// Mitsubishi GX Works2 project: PLC_7_27.11_watch   PLC: FX3G

// global labels: Global1
VAR_GLOBAL CONSTANT
  Const_flickers : REAL := 5;
END_VAR
VAR_GLOBAL
  SW_start_day AT X010 : BOOL;
  LI_active_day AT Y010 : BOOL;
  RE_init_org AT D1100 : REAL;
  RE_init_pml AT D1105 : REAL;
  RE_init_clm AT D1110 : REAL;
  RE_wash_org AT D1130 : REAL;
  RE_wash_pml AT D1135 : REAL;
  RE_wash_clm AT D1140 : REAL;
  RE_squeeze AT D1145 : REAL;
  RE_juice AT D1150 : REAL;
  RE_storage AT D1155 : REAL;
  SW_emeragnce AT X007 : BOOL;
  SW_start_wash AT X002 : BOOL;
  LI_active_wash AT Y005 : BOOL;
  SW_col_fruits AT X001 : BOOL;
  LI_active_col AT Y001 : BOOL;
  SW_start_squeeze AT X011 : BOOL;
  LI_flicker_1 AT Y002 : BOOL;
  LI_flicker_2 AT Y003 : BOOL;
  SW_qa AT X003 : BOOL;
END_VAR
VAR_GLOBAL CONSTANT
  Const_min_Range : INT := 1;
  Const_max_Range : INT := 5;
END_VAR
VAR_GLOBAL
  LI_qa AT Y004 : BOOL;
  Analog_output AT D8282 : REAL;
END_VAR
VAR_GLOBAL CONSTANT
  Const_ratio_2 : REAL := 2;
END_VAR
VAR_GLOBAL
  HL_3_sec_stop AT M0 : BOOL;
  HL_blink1 AT M1 : BOOL;
  HL_first_init AT M2 : BOOL;
END_VAR
VAR_GLOBAL CONSTANT
  Const_min_fruit : REAL := 1;
END_VAR
VAR_GLOBAL
  HL_min_fruit AT M3 : BOOL;
  HL_first_check AT M4 : BOOL;
END_VAR
VAR_GLOBAL CONSTANT
  Const_timer_3 : INT := 30;
END_VAR
VAR_GLOBAL
  TC_timer_3 AT TC3 : BOOL;
  TS_timer_3 AT TS3 : BOOL;
  HL_blink2 AT M5 : BOOL;
  HL_blink3 AT M6 : BOOL;
  TC_blink1 AT TC1 : BOOL;
  TS_blink1 AT TS1 : BOOL;
  TC_blink2 AT TC2 : BOOL;
  TS_blink2 AT TS2 : BOOL;
  TN_timer_3 AT TN3 : INT;
  TN_blink1 AT TN1 : INT;
  HL_stop_day AT M7 : BOOL;
  HL_start_wash AT M8 : BOOL;
  HL_active_day AT M9 : BOOL;
  RE_buffer AT D1170 : REAL;
END_VAR
VAR_GLOBAL CONSTANT
  Const_max_org : REAL := 50;
END_VAR
VAR_GLOBAL
  RE_half_amount AT D1175 : REAL;
  HL_end_station_1 AT M11 : BOOL;
  HL_reset_day AT M12 : BOOL;
  HL_start_squeeze AT M13 : BOOL;
  HL_blink_end AT M14 : BOOL;
  HL_end_station_3 AT M15 : BOOL;
  HL_end_station_2 AT M16 : BOOL;
  HL_end_station_4 AT M17 : BOOL;
  RE_analog_input AT D8201 : INT;
  HL_min_range AT M18 : BOOL;
  HL_max_range AT M19 : BOOL;
  HL_start_station_4 AT M20 : BOOL;
  RE_timer_generic AT D1185 : INT;
END_VAR
VAR_GLOBAL CONSTANT
  Const_timer_5 : INT := 50;
END_VAR
VAR_GLOBAL
  HL_help_check AT M21 : BOOL;
  HL_bad_test AT M22 : BOOL;
  CC_counter AT CC0 : BOOL;
END_VAR
VAR_GLOBAL CONSTANT
  Const_counter : INT := 2;
END_VAR
VAR_GLOBAL
  CS_counter AT CS0 : BOOL;
  HL_garbge AT M23 : BOOL;
  Analog_Input AT D8281 : INT;
  RE_div_to_normal AT D1190 : REAL;
END_VAR
VAR_GLOBAL CONSTANT
  Const_200 : INT := 200;
  Const_400 : INT := 400;
END_VAR
VAR_GLOBAL
  HL_check_wash1 AT M24 : BOOL;
  HL_check_wash2 AT M25 : BOOL;
  SW_start_donation AT X005 : BOOL;
  LI_donation1 AT Y006 : BOOL;
  RE_donation AT D1200 : REAL;
  RE_donation_org AT D1205 : INT;
  RE_donation_clm AT D1210 : INT;
  RE_donation_pml AT D1215 : INT;
  RE_donation_org_real AT D1220 : REAL;
  RE_donation_clm_real AT D1225 : REAL;
  RE_donation_pml_real AT D1230 : REAL;
END_VAR
VAR_GLOBAL CONSTANT
  Const_0 : REAL;
END_VAR
VAR_GLOBAL
  HL_donation_remain AT M26 : BOOL;
  LI_donation2 AT Y007 : BOOL;
END_VAR
VAR_GLOBAL CONSTANT
  Const_min_storage : INT := 150;
  Const_max_storage : INT := 300;
END_VAR
VAR_GLOBAL
  HL_end_station_0 AT M27 : BOOL;
END_VAR
VAR_GLOBAL CONSTANT
  Const_range_0 : REAL := 9472;
  Const_range_1 : REAL := 9475;
  Const_range_2 : REAL := 9476;
END_VAR
VAR_GLOBAL
  RE_range : ARRAY [0..2] OF BOOL;
  HL_storage_range0 AT M100 : BOOL;
  HL_storage_range1 AT M101 : BOOL;
  HL_storage_range2 AT M102 : BOOL;
  RE_storage_int AT D1232 : INT;
  HL_end_indicator_station_0 AT M103 : BOOL;
  CN_counter AT CN0 : INT;
END_VAR
VAR_GLOBAL CONSTANT
  Const_timer_03 : INT := 3;
  Const_ratio_2_modulo : INT := 2;
END_VAR

// task Task_01 (event TRUE, interval 0, priority 31): POU_01

PROGRAM POU_01
(* structured ladder/FBD written out as ST: instructions are called as NAME(EN, inputs, outputs); _pN, _eN, _tN stand for wires *)
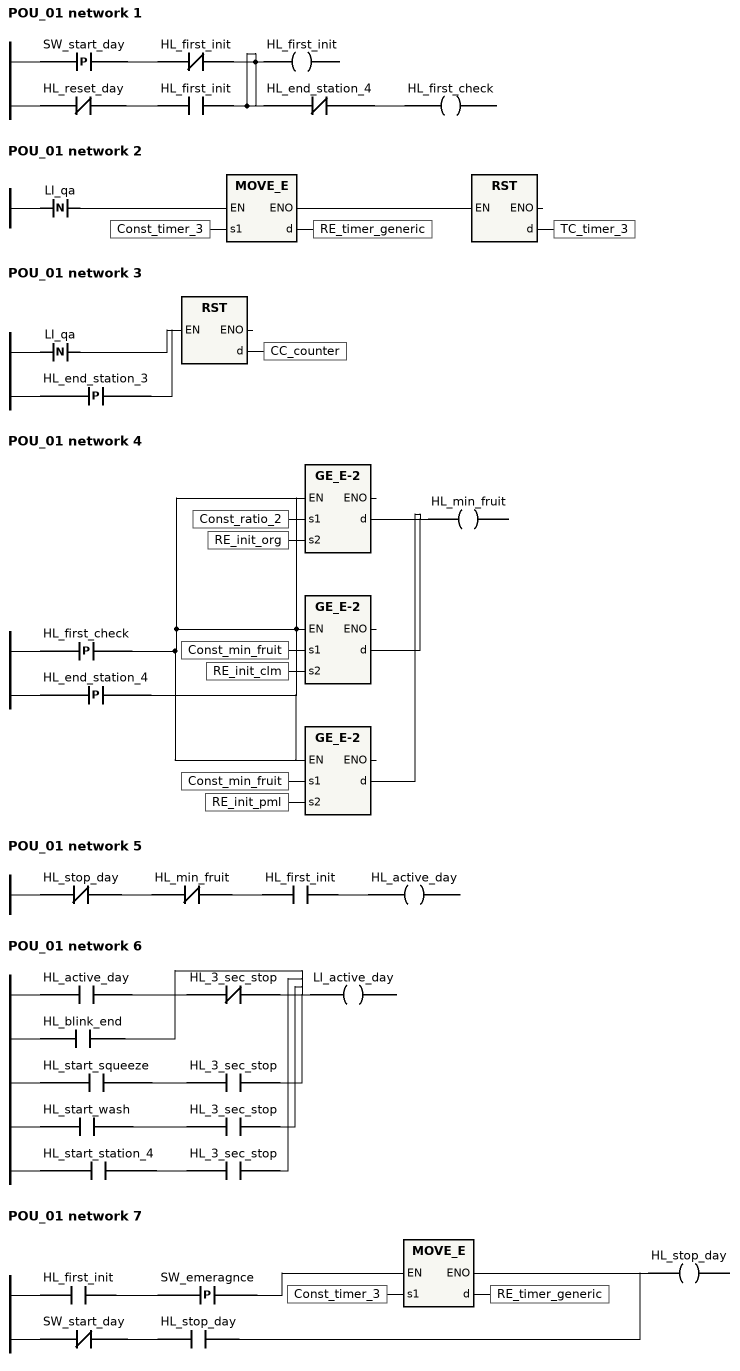
(* network 1 *)
_p1 := (LDP(TRUE, SW_start_day) AND NOT HL_first_init) OR (NOT HL_reset_day AND HL_first_init);
HL_first_init := _p1;
HL_first_check := _p1 AND NOT HL_end_station_4;
(* network 2 *)
_e1 := MOVE_E(LDF(TRUE, LI_qa), Const_timer_3, RE_timer_generic);
RST(_e1, TC_timer_3);
(* network 3 *)
RST(LDF(TRUE, LI_qa) OR LDP(TRUE, HL_end_station_3), CC_counter);
(* network 4 *)
_p1 := LDP(TRUE, HL_first_check) OR LDP(TRUE, HL_end_station_4);
GE_E(_p1, Const_ratio_2, RE_init_org, _t2);
GE_E(_p1, Const_min_fruit, RE_init_clm, _t3);
GE_E(_p1, Const_min_fruit, RE_init_pml, _t4);
HL_min_fruit := _t2 OR _t3 OR _t4;
(* network 5 *)
HL_active_day := NOT HL_stop_day AND NOT HL_min_fruit AND HL_first_init;
(* network 6 *)
LI_active_day := (HL_active_day AND NOT HL_3_sec_stop) OR HL_blink_end OR (HL_start_squeeze AND HL_3_sec_stop) OR (HL_start_wash AND HL_3_sec_stop) OR (HL_start_station_4 AND HL_3_sec_stop);
(* network 7 *)
_e1 := MOVE_E(HL_first_init AND LDP(TRUE, SW_emeragnce), Const_timer_3, RE_timer_generic);
HL_stop_day := _e1 OR (NOT SW_start_day AND HL_stop_day);
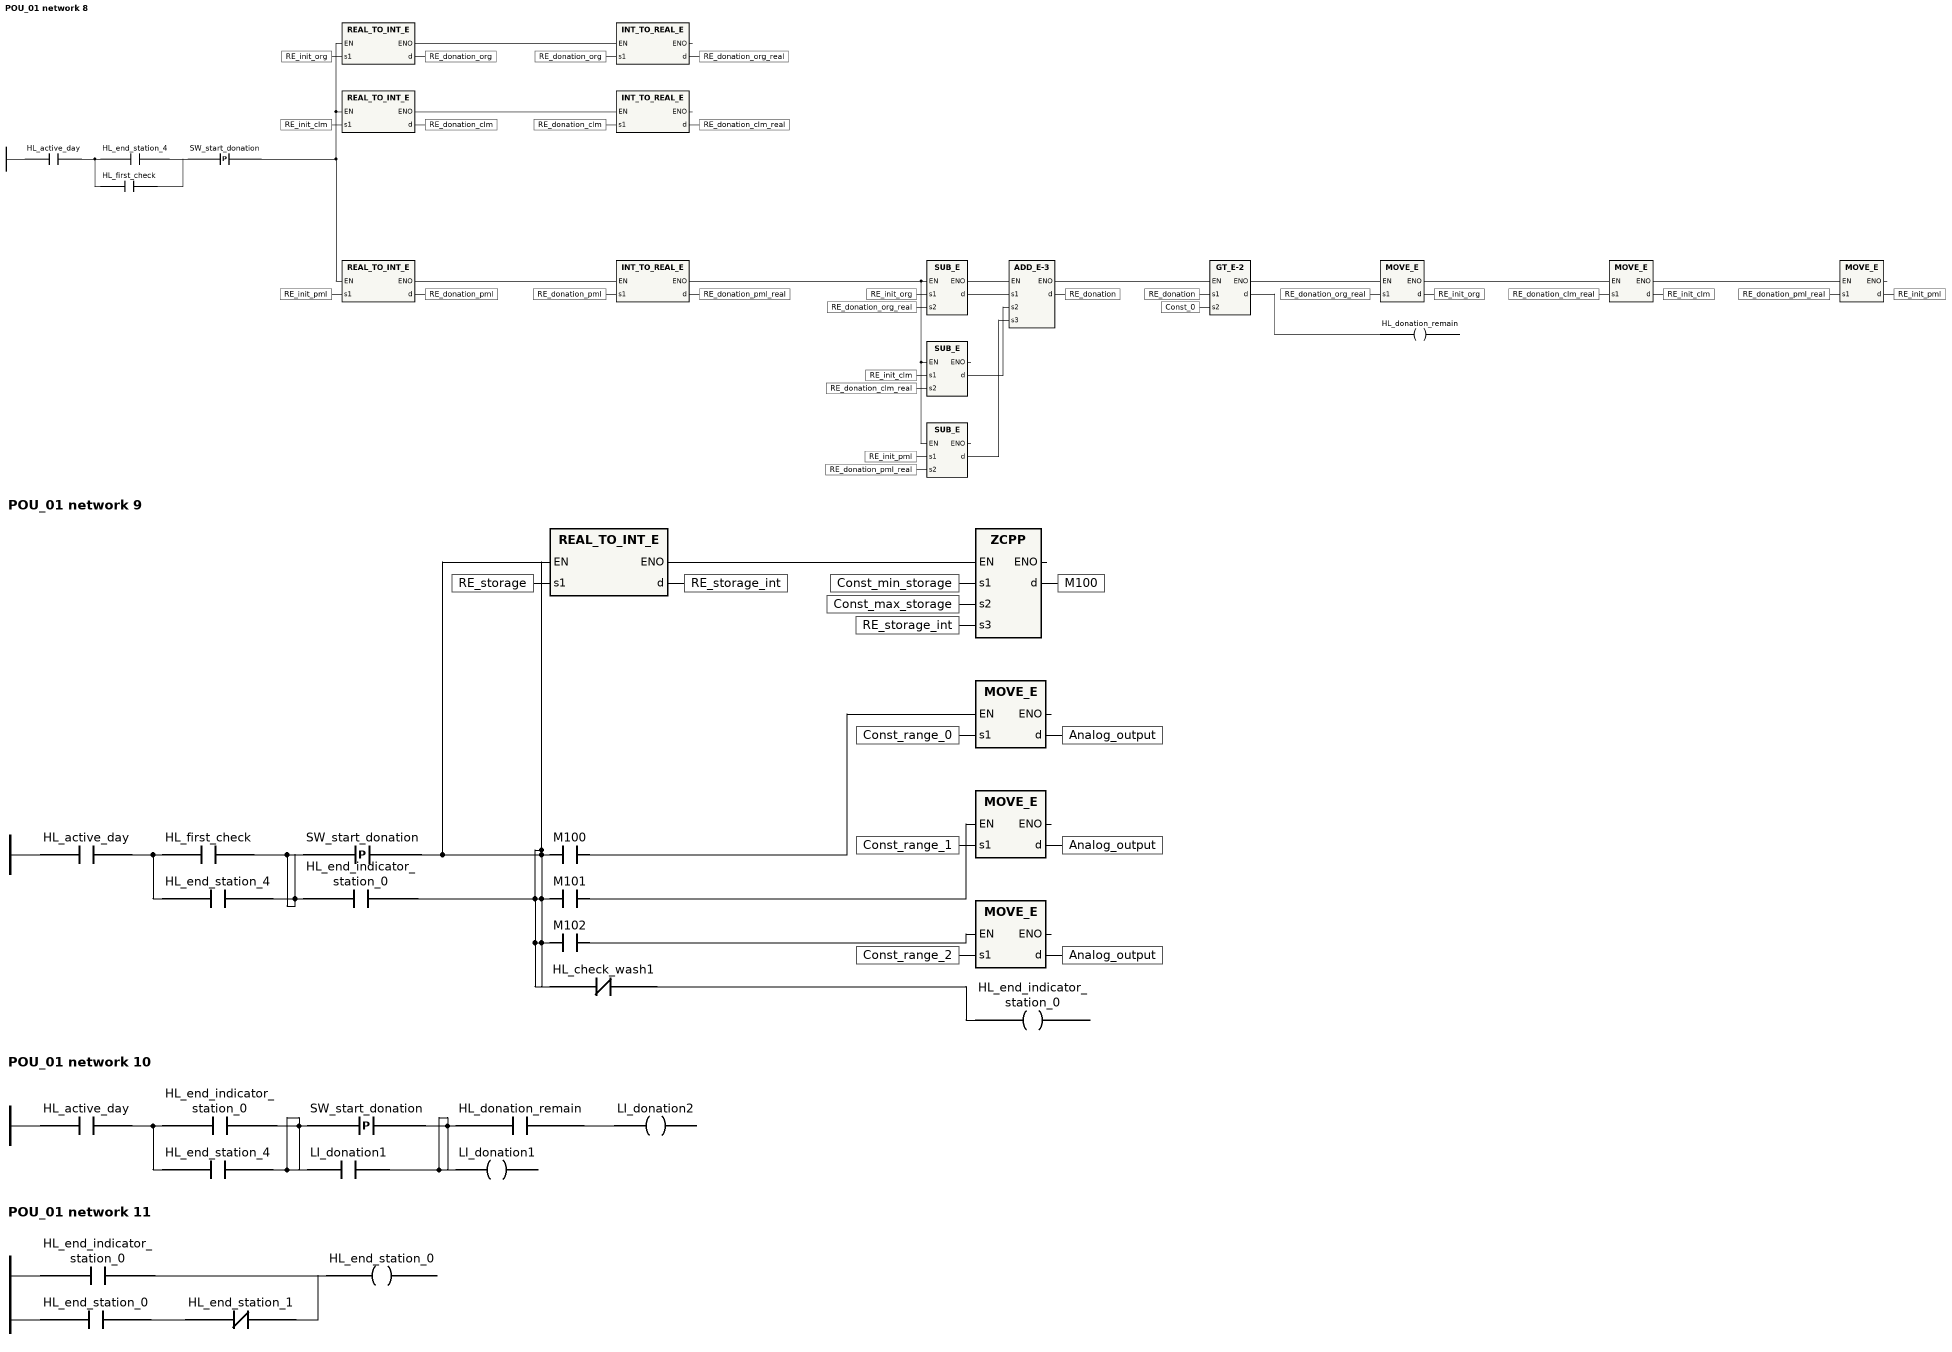
(* network 8 *)
_p1 := ((HL_active_day AND HL_end_station_4) OR (HL_active_day AND HL_first_check)) AND LDP(TRUE, SW_start_donation);
_e2 := REAL_TO_INT_E(_p1, RE_init_org, RE_donation_org);
INT_TO_REAL_E(_e2, RE_donation_org, RE_donation_org_real);
_e3 := REAL_TO_INT_E(_p1, RE_init_clm, RE_donation_clm);
INT_TO_REAL_E(_e3, RE_donation_clm, RE_donation_clm_real);
_e4 := REAL_TO_INT_E(_p1, RE_init_pml, RE_donation_pml);
_e5 := INT_TO_REAL_E(_e4, RE_donation_pml, RE_donation_pml_real);
_e7 := SUB_E(_e5, RE_init_org, RE_donation_org_real, _t6);
SUB_E(_e5, RE_init_clm, RE_donation_clm_real, _t8);
SUB_E(_e5, RE_init_pml, RE_donation_pml_real, _t9);
_e10 := ADD_E(_e7, _t6, _t8, _t9, RE_donation);
_e12 := GT_E(_e10, RE_donation, Const_0, _t11);
HL_donation_remain := _t11;
_e13 := MOVE_E(_e12, RE_donation_org_real, RE_init_org);
_e14 := MOVE_E(_e13, RE_donation_clm_real, RE_init_clm);
MOVE_E(_e14, RE_donation_pml_real, RE_init_pml);
(* network 9 *)
_p1 := (HL_active_day AND HL_first_check) OR (HL_active_day AND HL_end_station_4);
_p2 := (_p1 AND LDP(TRUE, SW_start_donation)) OR (_p1 AND HL_end_indicator_station_0);
_e3 := REAL_TO_INT_E(_p2, RE_storage, RE_storage_int);
ZCPP(_e3, Const_min_storage, Const_max_storage, RE_storage_int, M100);
MOVE_E(_p2 AND M100, Const_range_0, Analog_output);
MOVE_E(_p2 AND M101, Const_range_1, Analog_output);
MOVE_E(_p2 AND M102, Const_range_2, Analog_output);
HL_end_indicator_station_0 := _p2 AND NOT HL_check_wash1;
(* network 10 *)
_p1 := (HL_active_day AND HL_end_indicator_station_0) OR (HL_active_day AND HL_end_station_4);
_p2 := (_p1 AND LDP(TRUE, SW_start_donation)) OR (_p1 AND LI_donation1);
LI_donation2 := _p2 AND HL_donation_remain;
LI_donation1 := _p2;
(* network 11 *)
HL_end_station_0 := HL_end_indicator_station_0 OR (HL_end_station_0 AND NOT HL_end_station_1);
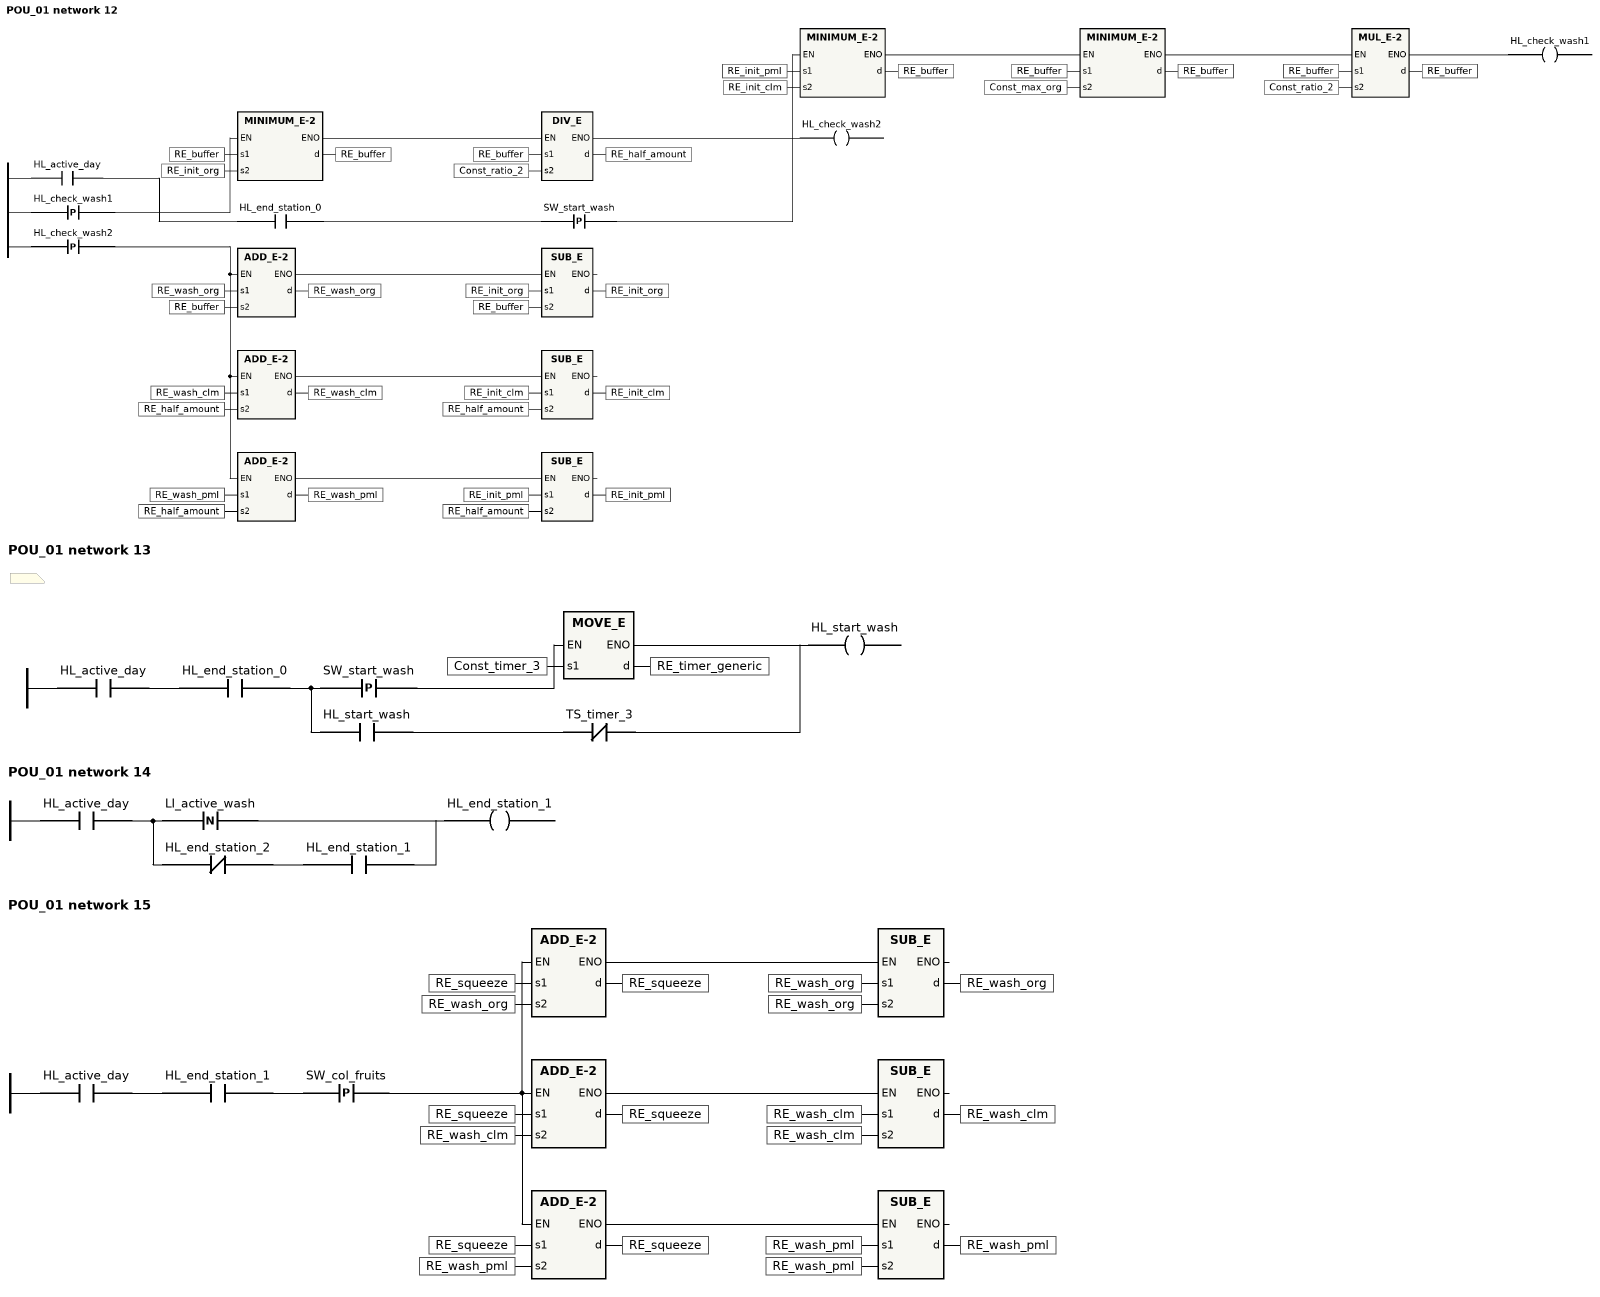
(* network 12 *)
_e1 := MINIMUM_E(HL_active_day AND HL_end_station_0 AND LDP(TRUE, SW_start_wash), RE_init_pml, RE_init_clm, RE_buffer);
_e2 := MINIMUM_E(_e1, RE_buffer, Const_max_org, RE_buffer);
_e3 := MUL_E(_e2, RE_buffer, Const_ratio_2, RE_buffer);
HL_check_wash1 := _e3;
_e4 := MINIMUM_E(LDP(TRUE, HL_check_wash1), RE_buffer, RE_init_org, RE_buffer);
_e5 := DIV_E(_e4, RE_buffer, Const_ratio_2, RE_half_amount);
HL_check_wash2 := _e5;
_p6 := LDP(TRUE, HL_check_wash2);
_e7 := ADD_E(_p6, RE_wash_org, RE_buffer, RE_wash_org);
SUB_E(_e7, RE_init_org, RE_buffer, RE_init_org);
_e8 := ADD_E(_p6, RE_wash_clm, RE_half_amount, RE_wash_clm);
SUB_E(_e8, RE_init_clm, RE_half_amount, RE_init_clm);
_e9 := ADD_E(_p6, RE_wash_pml, RE_half_amount, RE_wash_pml);
SUB_E(_e9, RE_init_pml, RE_half_amount, RE_init_pml);
(* network 13 *)
(*  *)
_p1 := HL_active_day AND HL_end_station_0;
_e2 := MOVE_E(_p1 AND LDP(TRUE, SW_start_wash), Const_timer_3, RE_timer_generic);
HL_start_wash := _e2 OR (_p1 AND HL_start_wash AND NOT TS_timer_3);
(* network 14 *)
HL_end_station_1 := (HL_active_day AND LDF(TRUE, LI_active_wash)) OR (HL_active_day AND NOT HL_end_station_2 AND HL_end_station_1);
(* network 15 *)
_p1 := HL_active_day AND HL_end_station_1 AND LDP(TRUE, SW_col_fruits);
_e2 := ADD_E(_p1, RE_squeeze, RE_wash_org, RE_squeeze);
SUB_E(_e2, RE_wash_org, RE_wash_org, RE_wash_org);
_e3 := ADD_E(_p1, RE_squeeze, RE_wash_clm, RE_squeeze);
SUB_E(_e3, RE_wash_clm, RE_wash_clm, RE_wash_clm);
_e4 := ADD_E(_p1, RE_squeeze, RE_wash_pml, RE_squeeze);
SUB_E(_e4, RE_wash_pml, RE_wash_pml, RE_wash_pml);
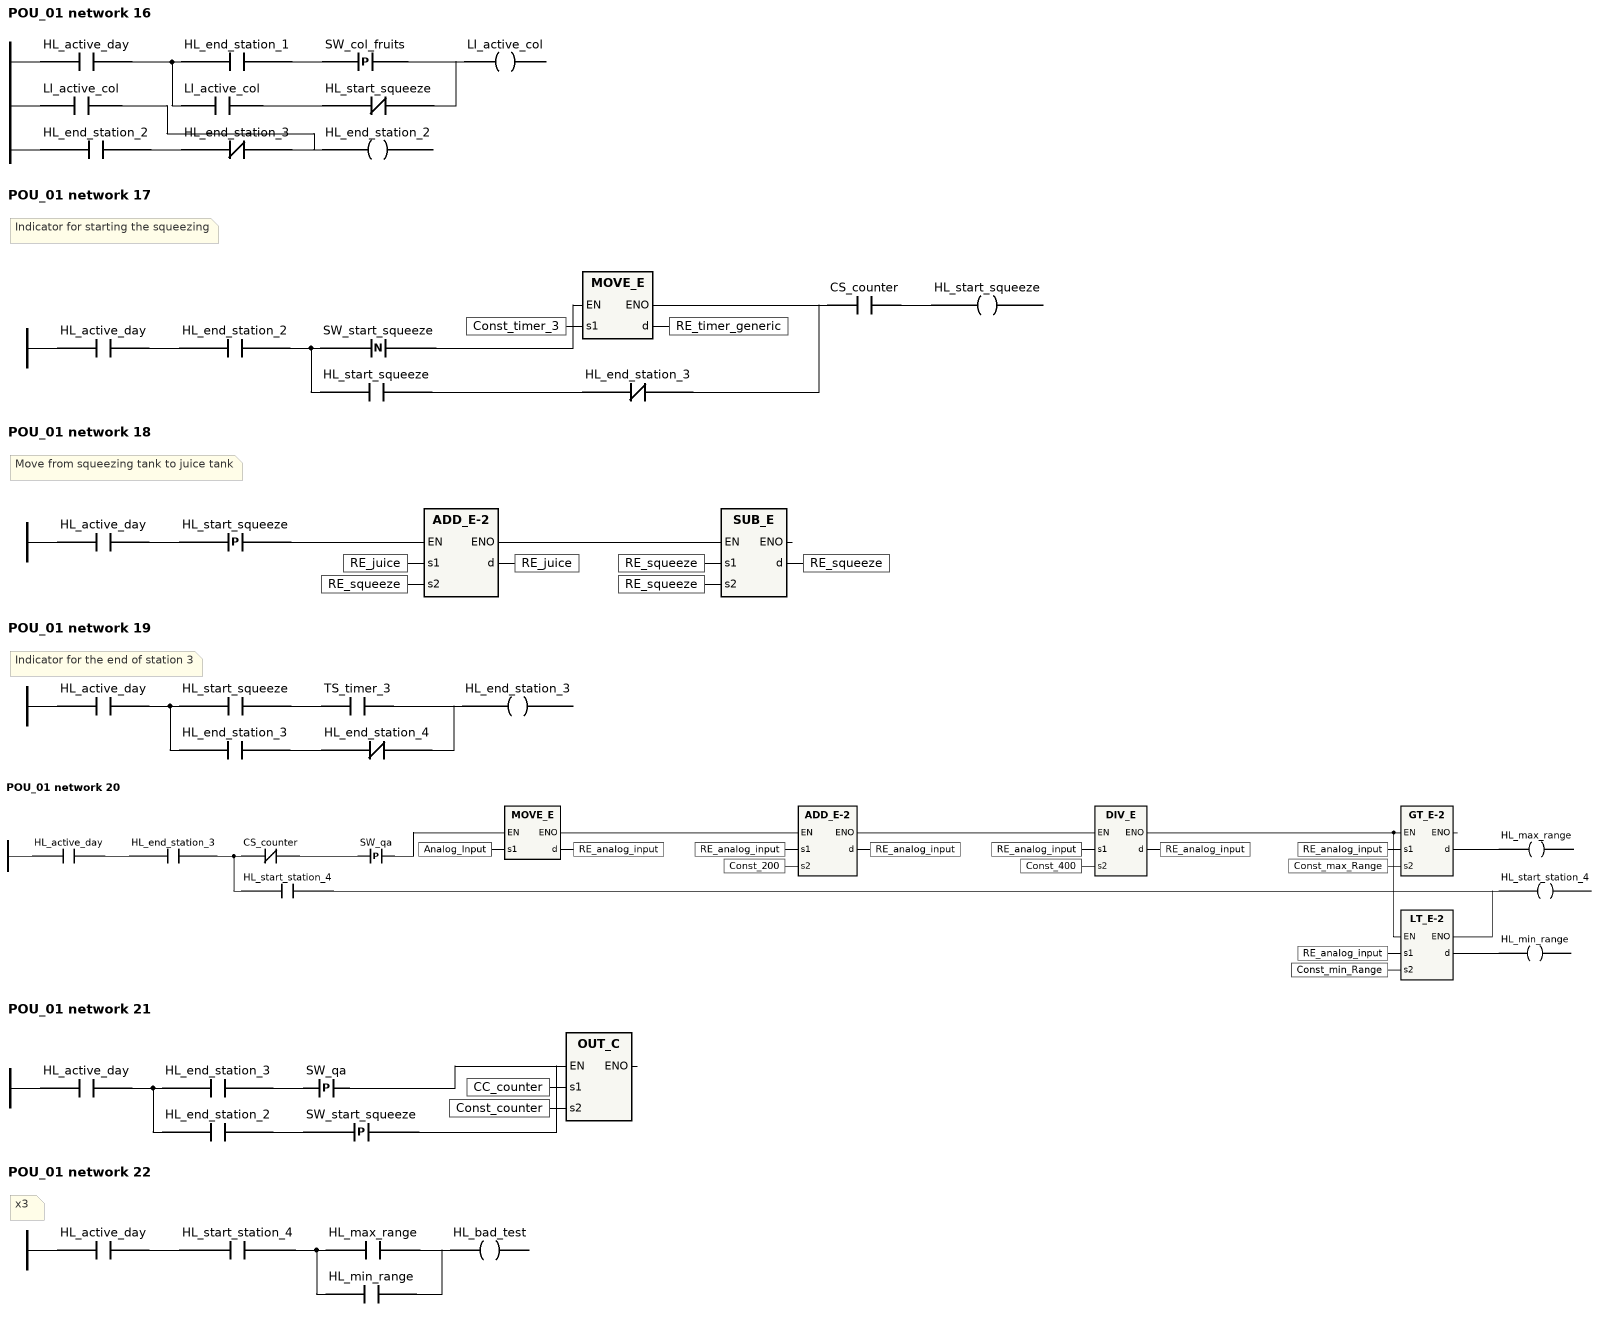
(* network 16 *)
LI_active_col := (HL_active_day AND HL_end_station_1 AND LDP(TRUE, SW_col_fruits)) OR (HL_active_day AND LI_active_col AND NOT HL_start_squeeze);
HL_end_station_2 := LI_active_col OR (HL_end_station_2 AND NOT HL_end_station_3);
(* network 17 *)
(* Indicator for starting the squeezing *)
_p1 := HL_active_day AND HL_end_station_2;
_e2 := MOVE_E(_p1 AND LDF(TRUE, SW_start_squeeze), Const_timer_3, RE_timer_generic);
HL_start_squeeze := (_e2 OR (_p1 AND HL_start_squeeze AND NOT HL_end_station_3)) AND CS_counter;
(* network 18 *)
(* Move from squeezing tank to juice tank *)
_e1 := ADD_E(HL_active_day AND LDP(TRUE, HL_start_squeeze), RE_juice, RE_squeeze, RE_juice);
SUB_E(_e1, RE_squeeze, RE_squeeze, RE_squeeze);
(* network 19 *)
(* Indicator for the end of station 3 *)
HL_end_station_3 := (HL_active_day AND HL_start_squeeze AND TS_timer_3) OR (HL_active_day AND HL_end_station_3 AND NOT HL_end_station_4);
(* network 20 *)
_p1 := HL_active_day AND HL_end_station_3;
_e2 := MOVE_E(_p1 AND NOT CS_counter AND LDP(TRUE, SW_qa), Analog_Input, RE_analog_input);
_e3 := ADD_E(_e2, RE_analog_input, Const_200, RE_analog_input);
_e4 := DIV_E(_e3, RE_analog_input, Const_400, RE_analog_input);
GT_E(_e4, RE_analog_input, Const_max_Range, _t5);
HL_max_range := _t5;
_e7 := LT_E(_e4, RE_analog_input, Const_min_Range, _t6);
HL_start_station_4 := _e7 OR (_p1 AND HL_start_station_4);
HL_min_range := _t6;
(* network 21 *)
OUT_C((HL_active_day AND HL_end_station_3 AND LDP(TRUE, SW_qa)) OR (HL_active_day AND HL_end_station_2 AND LDP(TRUE, SW_start_squeeze)), CC_counter, Const_counter);
(* network 22 *)
(* x3 *)
_p1 := HL_active_day AND HL_start_station_4;
HL_bad_test := (_p1 AND HL_max_range) OR (_p1 AND HL_min_range);
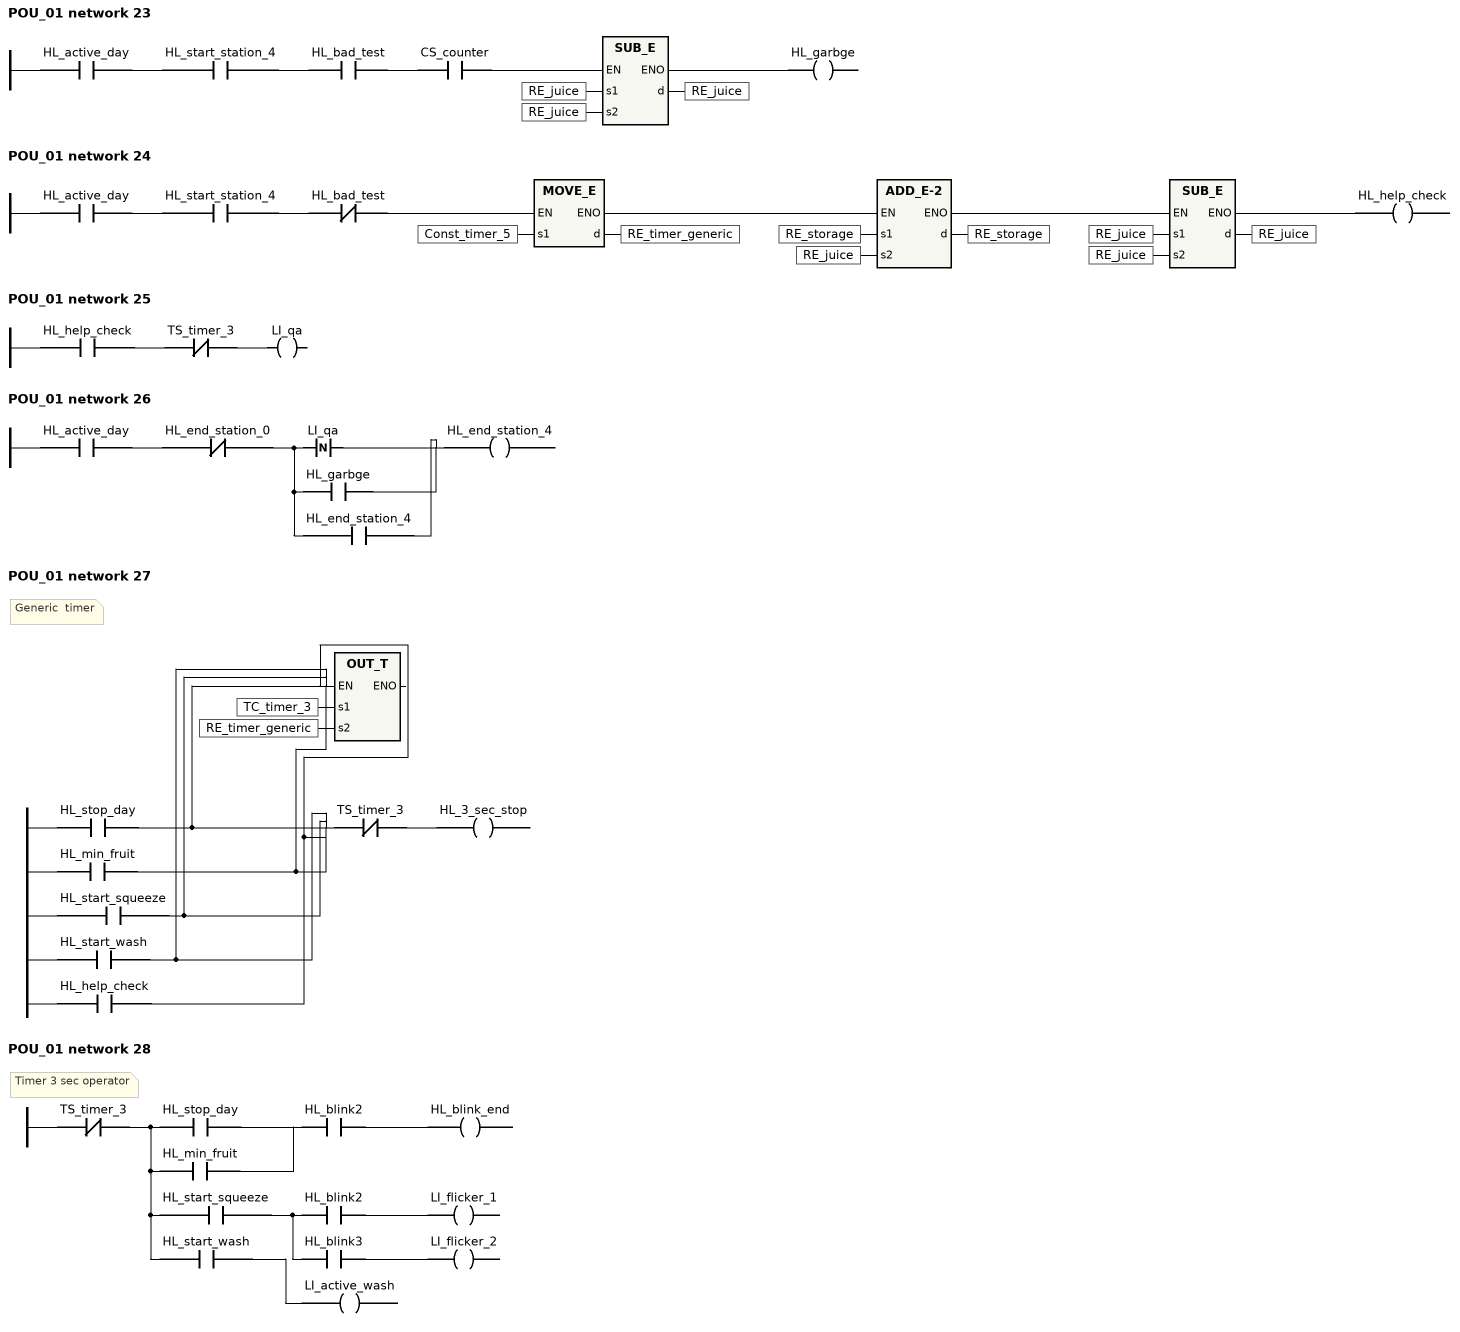
(* network 23 *)
_e1 := SUB_E(HL_active_day AND HL_start_station_4 AND HL_bad_test AND CS_counter, RE_juice, RE_juice, RE_juice);
HL_garbge := _e1;
(* network 24 *)
_e1 := MOVE_E(HL_active_day AND HL_start_station_4 AND NOT HL_bad_test, Const_timer_5, RE_timer_generic);
_e2 := ADD_E(_e1, RE_storage, RE_juice, RE_storage);
_e3 := SUB_E(_e2, RE_juice, RE_juice, RE_juice);
HL_help_check := _e3;
(* network 25 *)
LI_qa := HL_help_check AND NOT TS_timer_3;
(* network 26 *)
_p1 := HL_active_day AND NOT HL_end_station_0;
HL_end_station_4 := (_p1 AND LDF(TRUE, LI_qa)) OR (_p1 AND HL_garbge) OR (_p1 AND HL_end_station_4);
(* network 27 *)
(* Generic  timer *)
_p1 := HL_stop_day OR HL_min_fruit OR HL_start_squeeze OR HL_start_wash OR HL_help_check;
OUT_T(_p1, TC_timer_3, RE_timer_generic);
HL_3_sec_stop := _p1 AND NOT TS_timer_3;
(* network 28 *)
(* Timer 3 sec operator *)
_p1 := NOT TS_timer_3;
HL_blink_end := ((_p1 AND HL_stop_day) OR (_p1 AND HL_min_fruit)) AND HL_blink2;
_p2 := _p1 AND HL_start_squeeze;
LI_flicker_1 := _p2 AND HL_blink2;
LI_flicker_2 := _p2 AND HL_blink3;
LI_active_wash := _p1 AND HL_start_wash;
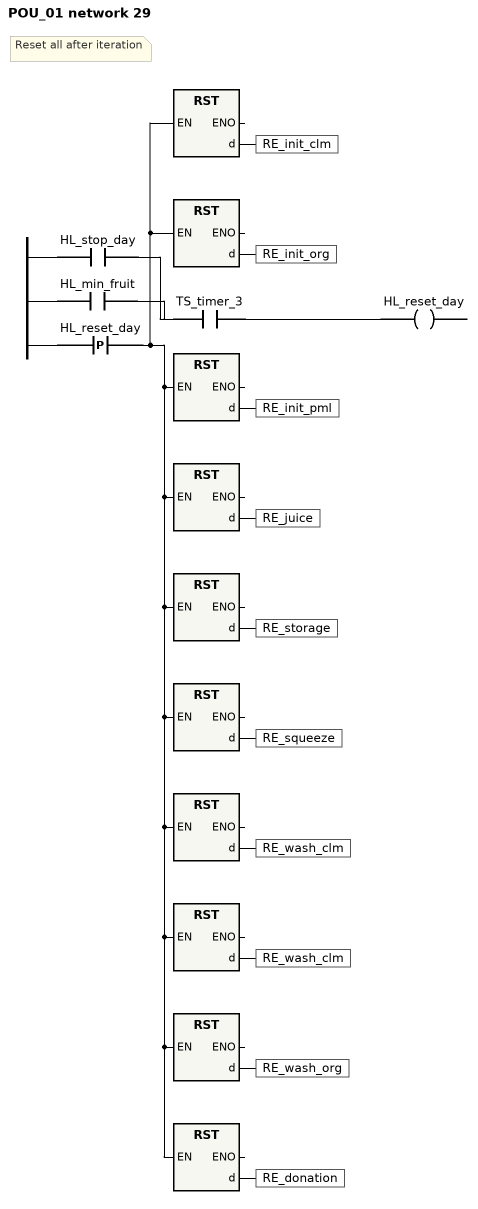
(* network 29 *)
(* Reset all after iteration *)
HL_reset_day := (HL_stop_day OR HL_min_fruit) AND TS_timer_3;
_p1 := LDP(TRUE, HL_reset_day);
RST(_p1, RE_init_clm);
RST(_p1, RE_init_org);
RST(_p1, RE_init_pml);
RST(_p1, RE_juice);
RST(_p1, RE_storage);
RST(_p1, RE_squeeze);
RST(_p1, RE_wash_clm);
RST(_p1, RE_wash_clm);
RST(_p1, RE_wash_org);
RST(_p1, RE_donation);
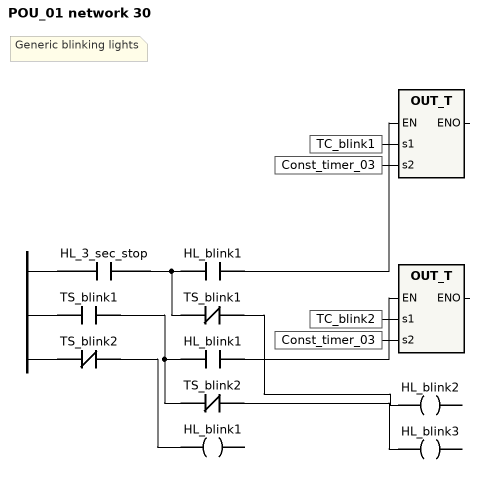
(* network 30 *)
(* Generic blinking lights *)
OUT_T(HL_3_sec_stop AND HL_blink1, TC_blink1, Const_timer_03);
HL_blink2 := HL_3_sec_stop AND NOT TS_blink1;
OUT_T(TS_blink1 AND HL_blink1, TC_blink2, Const_timer_03);
HL_blink3 := TS_blink1 AND NOT TS_blink2;
HL_blink1 := NOT TS_blink2;
END_PROGRAM
